// TIA Portal V16 export
// export: Created 2022-04-16T09:29:33.5655025Z, ExportSetting WithDefaults, DisplayName Totally Integrated Automation Portal, DisplayVersion V16 Update 3, DisplayName TIA Portal Version Control Interface, DisplayVersion V16 Update 2, DisplayName TIA Portal Openness, DisplayVersion V16 Update 3, DisplayName STEP 7 Professional, DisplayVersion V16 Update 3, DisplayName STEP 7 Safety, DisplayVersion V16, DisplayName WinCC Professional, DisplayVersion V16 Update 3
VAR_GLOBAL   // PLC tag table "PAL_TestFC02001"
   FIC101_RAW AT %MW100 : Int;   // FIC101 - Instrument Simulation - RAW SIGNAL
   FIC101_FLT AT %M110.0 : Bool;   // FIC101 - Instrument Simulation - EXTERNAL FAULT
END_VAR
